KUKA KRL data list: Prog.dat

&ACCESS RVO
DEFDAT  Init PUBLIC
DECL POS P1={X 0.0,Y 0.0,Z 0.0,A 0.0,B 0.0,C 0.0,S 6} ; pozice nad zasobnikem
DECL POS P2={X 0.0,Y 0.0,Z 0.0,A 0.0,B 0.0,C 0.0,S 6} ; bezpecna pozic
DECL POS P3={X 0.0,Y 0.0,Z 0.0,A 0.0,B 0.0,C 0.0,S 6} ; pozice nad kytkou

DECL INT leg_x_base = 0 ;
DECL INT leg_y_base = 0 ;
DECL INT stalk = 0 ;

DECL REAL safe = 0 ;
DECL REAL very_safe = 0 ;
DECL REAL x_pitch = 0 ;
DECL REAL y_pitch = 0 ;
DECL REAL z_pitch = 0 ;
DECL REAL x_base = 0 ;
DECL REAL y_base = 0 ;
ENDDAT
